ABB RAPID module: 001873CB

MODULE Module1
	CONST robtarget Target_10:=[[710.302,-50.687,666.042],[0,1,0,0],[-1,0,1,0],[9E+09,9E+09,9E+09,9E+09,9E+09,9E+09]];
	CONST robtarget Target_20:=[[760.301980587,-50.686989693,756.042035513],[-0.000000033,1,-0.000000027,0.000000018],[-1,-1,1,0],[9E+09,9E+09,9E+09,9E+09,9E+09,9E+09]];
	PROC Path_10()
	    MoveL Target_10,v1000,z100,Mano_de_Juan\WObj:=wobj0;
	    SetDO ActivaMano_Juan,1;
	    MoveL Target_20,v1000,z100,Mano_de_Juan\WObj:=wobj0;
	ENDPROC
ENDMODULE
